// TIA Portal V20 export
DATA_BLOCK "CELL"   // DB120
{ S7_Optimized_Access := 'FALSE' }
VERSION : 0.1
// stored: AutoNumber false, DBAccessibleFromOPCUA true, DBAccessibleFromWebserver true, IsOnlyStoredInLoadMemory false, IsWriteProtectedInAS false
   VAR RETAIN
      Count : UInt;
      Cell : Array["CELL_MIN".."CELL_MAX"] of "LGR_Cell_Info";
   END_VAR
BEGIN
END_DATA_BLOCK
